Universal Robots PolyScope program: LearningByDemo.urp

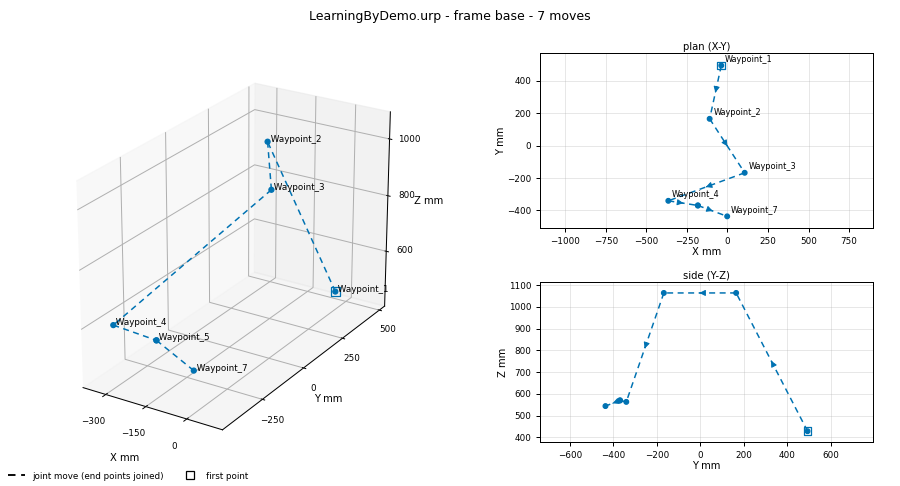
[picture p0: tool path of LearningByDemo.urp in frame base, 7 of 7 moves have a stored position in this frame; points joined in program order, loops and branches not executed]
Program ash333 (installation=SSR directory=/programs createdIn=5.9.1.1031110 lastSavedIn=5.9.1.1031110 robotSerialNumber=20195500561)
Calibrated DH parameters: a=[0.000135, -0.404407, -0.388607, 0, 0.000082, 0]; d=[0.162518, -89.171881, 146.306543, -57.001371, 0.099639, 0.099545]; alpha=[1.570833, 0.001462, -0.000956, 1.570431, -1.5702, 0]; deltaTheta=[0, -0.311794, 6.455277, 0.139702, 0.000002, 0]
Robot Program (runOnlyOnce=true)
  Wait Sleep waitTime=0.3
Event  expression=dockbut≟ True
  MoveJ speed 60 deg/s, acceleration 80 deg/s^2 (useActiveTCP=true positionType=JointAngles) feature=Base
    Waypoint Waypoint_1: motionParameters(blendRadius=0.05); TCP in base x=-38.007 y=493.637 z=428.017 mm, rx=-3.0042 ry=-0.2675 rz=0.0904 rad; joints [-102.251, -92.82, 103.16, -106.082, -84.688, 337.773] deg
      Until REACHED_WAYPOINT (allowActions=true)
        MoveJ speed 60 deg/s, acceleration 80 deg/s^2 (useActiveTCP=true positionType=JointAngles) feature=Base
          Waypoint Waypoint_2: TCP in base x=-109.659 y=165.145 z=1064.137 mm, rx=-1.6303 ry=-0.2154 rz=-0.3851 rad; joints [-102.162, -95.622, 16.649, -97.549, -84.694, 337.742] deg
            Until REACHED_WAYPOINT (allowActions=true)
              MoveJ speed 60 deg/s, acceleration 80 deg/s^2 (useActiveTCP=true positionType=JointAngles) feature=Base
                Waypoint Waypoint_3: TCP in base x=106.261 y=-167.575 z=1064.087 mm, rx=0.2495 ry=-2.0455 rz=1.8744 rad; joints [76.687, -95.607, 16.65, -97.545, -84.692, 337.74] deg
                  Until REACHED_WAYPOINT (allowActions=true)
                    MoveJ speed 60 deg/s, acceleration 80 deg/s^2 (useActiveTCP=true positionType=JointAngles) feature=Base
                      Waypoint Waypoint_4: motionParameters(blendRadius=0.05); TCP in base x=-364.427 y=-340.347 z=562.872 mm, rx=-0.4242 ry=-1.3744 rz=1.4466 rad; joints [26.539, -83.766, 105.538, -217.952, -84.694, 337.74] deg
                        Until REACHED_WAYPOINT (allowActions=true)
                          MoveJ speed 60 deg/s, acceleration 80 deg/s^2 (useActiveTCP=true positionType=JointAngles) feature=Base
                            Waypoint Waypoint_5: motionParameters(blendRadius=0); TCP in base x=-182.232 y=-369.118 z=569.675 mm, rx=-1.6431 ry=1.4283 rz=-1.8393 rad; joints [31.749, -83.807, 98.114, -210.431, 31.166, 337.733] deg
                              Until REACHED_WAYPOINT (allowActions=true)
                                MoveJ speed 60 deg/s, acceleration 80 deg/s^2 (useActiveTCP=true positionType=JointAngles) feature=Base
                                  Waypoint Waypoint_6: motionParameters(blendRadius=0); TCP in base x=-182.212 y=-369.115 z=569.699 mm, rx=0.7015 ry=1.5649 rz=-0.1049 rad; joints [31.749, -83.809, 98.11, -210.445, 31.157, 124.036] deg
                                    Until REACHED_WAYPOINT (allowActions=true)
                                      MoveJ speed 60 deg/s, acceleration 80 deg/s^2 (useActiveTCP=true positionType=JointAngles) feature=Base
                                        Waypoint Waypoint_7: motionParameters(blendRadius=0.05); TCP in base x=-1.532 y=-436.158 z=543.61 mm, rx=-1.684 ry=-1.7535 rz=1.2805 rad; joints [-60.214, -169.167, 98.095, -210.457, 31.164, 124.041] deg
                                          Until REACHED_WAYPOINT (allowActions=true)
                                            Halt
